// SIMATIC S7-200 SMART project (STEP 7-Micro/WIN SMART), CPU SR40

ORGANIZATION_BLOCK 主程序:OB1
TITLE=程序注释
BEGIN
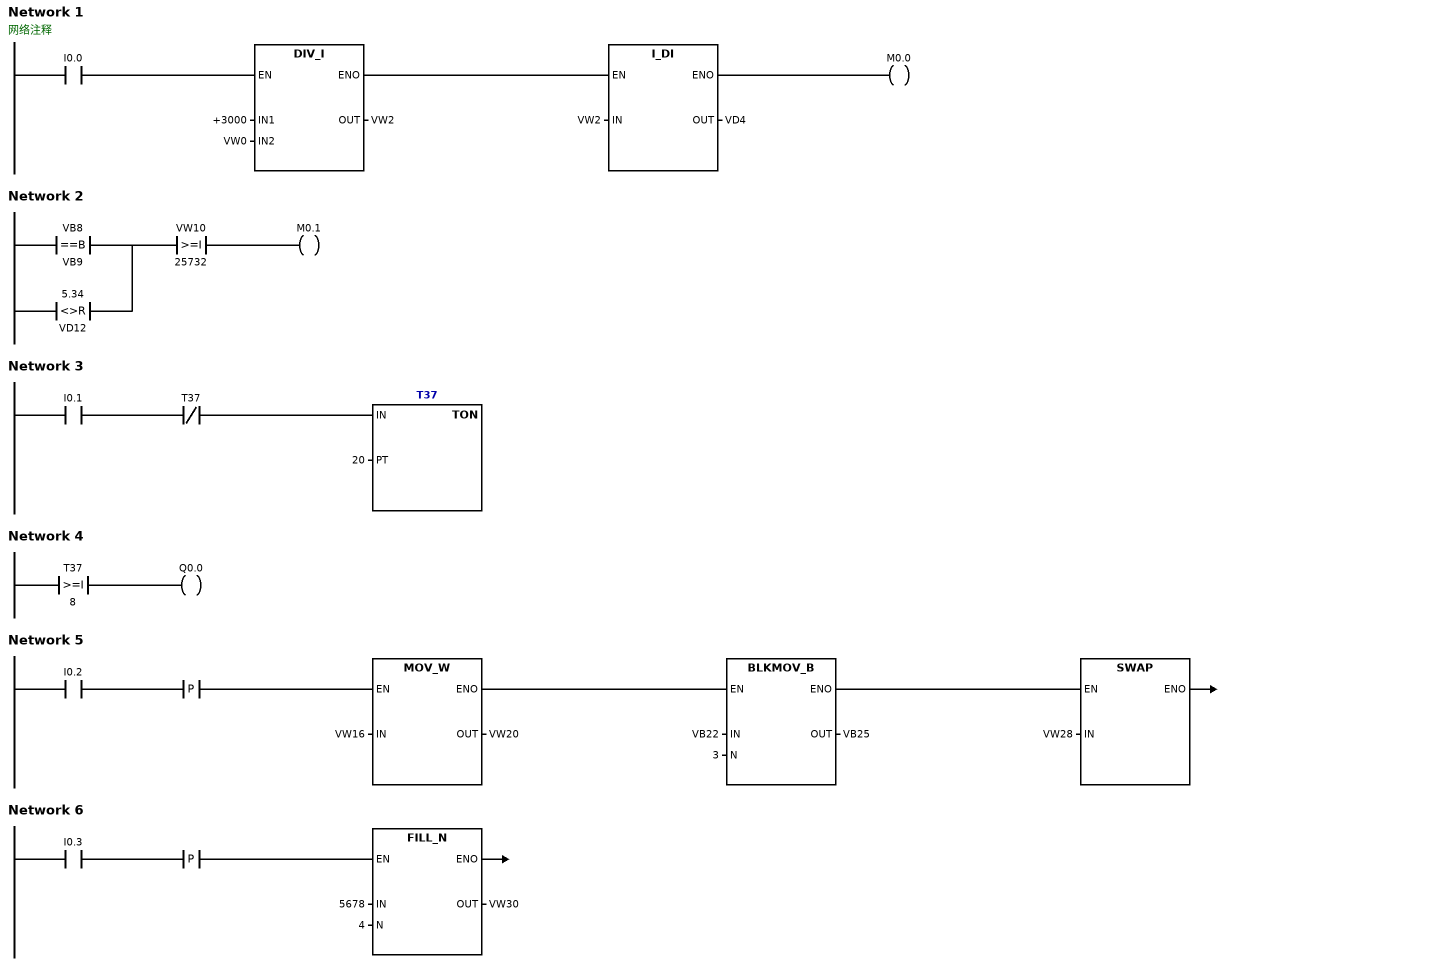
Network 1
// 网络注释
LD     I0.0
MOVW   +3000, VW2
AENO
/I     VW0, VW2
AENO
ITD    VW2, VD4
AENO
=      M0.0
Network 2
LDB=   VB8, VB9
OR<>   5.34, VD12
AW>=   VW10, 25732
=      M0.1
Network 3
LD     I0.1
AN     T37
TON    T37, 20
Network 4
LDW>=  T37, 8
=      Q0.0
Network 5
LD     I0.2
EU
MOVW   VW16, VW20
AENO
BMB    VB22, VB25, 3
AENO
SWAP   VW28
Network 6
LD     I0.3
EU
FILL   5678, VW30, 4
END_ORGANIZATION_BLOCK
